# EPICS substitutions: evrSupport/Db/ioc/IOC-IN20-LS13evr.substitutions
#==============================================================================
#
# Abs:  LCLS EVR IOC records for IN20 LS13
#
# Name: IOC-IN20-LS13evr.substitutions
#
#==============================================================================
#
file evrAMXX.db
{
pattern { DEVICE        }
	{ EVR:IN20:LS13 }
}
